FUNCTION_BLOCK GetInstancePathAndName (* Function block to retrieve instance path and instance name from the runtime *)
  PACKAGE eclipse4diac::utils;
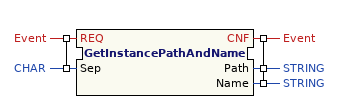
  EVENT_INPUT
    REQ WITH Sep; (* Service Request *)
  END_EVENT
  EVENT_OUTPUT
    CNF WITH Path, Name; (* Confirmation of Requested Service *)
  END_EVENT
  VAR_INPUT
    Sep : CHAR := '/'; (* Separator character for the output path generated by this FB *)
  END_VAR
  VAR_OUTPUT
    Path : STRING; (* Instance path of this FB *)
    Name : STRING; (* Instance name of this FB *)
  END_VAR
END_FUNCTION_BLOCK
